// TIA Portal V16 program export: 1 tag tables, 0 data types, 0 data blocks, 1 code blocks (in call order from the OBs), 0 instance data blocks

VAR_GLOBAL   // PLC tag table "Default tag table"
   START AT %I0.0 : Bool;
   STOP AT %I0.1 : Bool;
   AUTO AT %I0.2 : Bool;
   RESET AT %I0.3 : Bool;
   SORTER_EXTENDED AT %I1.0 : Bool;
   "PARTS_IN _STORAGE" AT %I1.1 : Bool;
   SORTER AT %Q5.0 : Bool;
   CONVEYER AT %Q5.1 : Bool;
END_VAR

ORGANIZATION_BLOCK "Main"   // OB1, LAD, ProgramCycle
TITLE = "Main Program Sweep (Cycle)"
{ S7_Optimized_Access := 'TRUE' }
VERSION : 0.1
// stored: AutoNumber true, IsIECCheckEnabled false, SetENOAutomatically false
   VAR_INPUT
      Initial_Call : Bool;   // Initial call of this OB
      Remanence : Bool;   // =True, if remanent data are available
   END_VAR
BEGIN
END_ORGANIZATION_BLOCK
